{attribute 'qualified_only'}
//General control ascii charachters
VAR_GLOBAL CONSTANT
    STX	  : BYTE := 16#02; //Start of text
    ETX   : BYTE := 16#03; //End of text
    Space : BYTE := 16#20; //Space
	CR	  : BYTE := 16#0D; //Carriage return
	LF	  : BYTE := 16#0A; //Line feed
END_VAR

(* stored: Version 1.1.0.1, ProductVersion 3.1.4020.12
   GVL NTO_LibraryAscii: Id {9b377c13-9786-42f3-985c-d9af4c11aa90} *)
